FUNCTION_BLOCK FB_Flash
VAR_INPUT
	bEnable		: BOOL;
	tInterval	: TIME;
END_VAR
VAR_OUTPUT
	Q			: BOOL;
END_VAR
VAR
	tWait		: TON;
END_VAR


tWait(IN:= bEnable AND NOT tWait.Q  , PT:= tInterval);

IF bEnable THEN
	IF tWait.ET > (tInterval / 2) THEN
		Q	:= TRUE;
	ELSE
		Q	:= FALSE;
	END_IF
ELSE
	Q	:= FALSE;
END_IF

END_FUNCTION_BLOCK

(* stored: Version 1.1.0.1, ProductVersion 3.1.4022.6
   POU FB_Flash: Id {0d1d5e3f-6281-46ec-aa52-6b61ae3620f4}, SpecialFunc None *)
